Staubli VAL3: saveIt.pgx

program saveIt(bool& x_bSave[])
  local string l_sMessage
  local num l_nResult
  local string l_sEmpty
begin
  // unselect ALL
  call unSelectItem()

  // do the onSave trajtype
  l_sEmpty=""
  call trajType:onSave(l_sEmpty)
  logMsg("[KERNEL] INTERFACE:Save the trajectory "+saveData:sTrajTypeUsing+": "+sTrajName)
  x_bSave=false
  sItems[0]="saved"
  call language:message(l_sMessage,-4)
  call use:timerDialog(l_sMessage,1)
end
